FUNCTION TryConvert_USINT_TO_DATE : BOOL
VAR_INPUT
	in : USINT;
	out : REFERENCE TO DATE;
END_VAR

out := USINT_TO_DATE(in);
TryConvert_USINT_TO_DATE := TRUE;

END_FUNCTION

(* stored: Version 1.1.0.1, ProductVersion 3.1.4024.12
   POU TryConvert_USINT_TO_DATE: Id {c93253d1-f83f-4cc9-b20c-a2b44d76190e}, SpecialFunc None *)
